PROGRAM PRG_LVCP2_Group7
VAR
    // Function Block Instance
    fbContactor: FB_ContactorControl;

    // Contactor 1 IO Structure  
    stContactor_IO: ST_ContactorIO;
    
    // Başlangıç konfigürasyonu için flag
    bContactorInitDone: BOOL := FALSE;
    bCapacitorInitDone: BOOL := FALSE;	
END_VAR



	M_Contactor();
	
	M_Capacitor();

METHOD M_Capacitor : BOOL
VAR
    nGroupIndex : INT;
END_VAR

nGroupIndex := 6;  // Grup 7 için index

IF NOT bCapacitorInitDone THEN
    // Grup 7 değerlerini ata
    GVL_LVCP2.astCompensationGroups[nGroupIndex].rPower := 25.0;
    GVL_LVCP2.astCompensationGroups[nGroupIndex].rVoltage := 450.0;
    GVL_LVCP2.astCompensationGroups[nGroupIndex].nQuantity := 2;
    GVL_LVCP2.astCompensationGroups[nGroupIndex].sTagPrefix := '+EP7-34C1';
    GVL_LVCP2.astCompensationGroups[nGroupIndex].sProductCode := 'ENT.CXD-450-25';
    
    bCapacitorInitDone := TRUE;
END_IF

// Grup 7 aktif durumu
GVL_LVCP2.abGroupActive[nGroupIndex] := stContactor_IO.bFeedback;

M_Capacitor := TRUE;
END_METHOD

METHOD M_Contactor : BOOL
VAR_INPUT
END_VAR
IF NOT bContactorInitDone THEN
    // Konfigürasyon parametreleri
    GVL_LVCP2.stGroup7_ContactorHMI.stConfig.sProjectCode := '+EP7-35K1';
    GVL_LVCP2.stGroup7_ContactorHMI.stConfig.sProductCode := 'ABB 1SFL447001R1311';
    GVL_LVCP2.stGroup7_ContactorHMI.stConfig.rRatedCurrent := 150.0;
    GVL_LVCP2.stGroup7_ContactorHMI.stConfig.rRatedVoltage := 1000.0;
    GVL_LVCP2.stGroup7_ContactorHMI.stConfig.nPhaseCount := 3;
    GVL_LVCP2.stGroup7_ContactorHMI.stConfig.tFeedbackDelay := T#500MS;
    GVL_LVCP2.stGroup7_ContactorHMI.stConfig.tWeldedDelay := T#2S;
    GVL_LVCP2.stGroup7_ContactorHMI.stConfig.dwOperationLimit := 100000;
    
    // Başlangıç bakım sayacı
    GVL_LVCP2.stGroup7_ContactorHMI.stStatistics.dwRemainingOperations := GVL_LVCP2.stGroup7_ContactorHMI.stConfig.dwOperationLimit;
    
    bContactorInitDone := TRUE;
END_IF

// Function Block Çağrısı
fbContactor(
    // Fiziksel Girişler
    bFeedback := stContactor_IO.bFeedback,
    bPLCControl := stContactor_IO.bPLCControl,
    
    // Güvenlik Girişleri
    bSafetyLoop := GVL_Alarm.bSafetyLoop,
    bInterlock := FALSE,
    
    // Sistem Girişleri
    bMasterReset := GVL_Alarm.bMasterReset,
    
    // HMI Bağlantısı
    stHMI := GVL_LVCP2.stGroup7_ContactorHMI,
    
    // Fiziksel Çıkış
    bOutput => stContactor_IO.bOutput
);

M_Contactor := TRUE;
END_METHOD

END_PROGRAM

(* stored: Version 1.1.0.1, ProductVersion 3.1.4024.14
   POU PRG_LVCP2_Group7: Id {3db08680-2685-41c8-8f1a-e817d7336a17}, SpecialFunc None
   Method M_Capacitor: Id {433c4584-7e5f-405f-a33f-fd21fb9b1f6f}
   Method M_Contactor: Id {a820ff8f-ea54-4d3e-8d5c-68f9b0593e77} *)
